// TIA Portal V21 export
TYPE "LAxisCtrl_typeGearOutCamOut"
TITLE = LAxisCtrl_typeGearOutCamOut
// Support: tech.team.motioncontrol@siemens.com
   STRUCT
      slavePosition : LReal := 0.0;   // Stop position of following axis
      syncProfileReference : DInt := 1;   // Type of desynchronization (0: Desynchronize using dynamic behavior; 1: Desynchronize using leading value distance; 5: Cancel only a pending gearing / camming)
      masterStopDistance : LReal := 0.0;   // Leading value distance when "SyncProfileReference" = 1
      deceleration : LReal := -1.0;   // Deceleration for desynchronization (Value > 0.0: The specified value is used; Value = 0.0: Not permitted; Value < 0.0: Use of the default value configured in the technology object) when "SyncProfileReference" = 0
      jerk : LReal := -1.0;   // Jerk for desynchronization (Value > 0.0: Smooth velocity profile, the specified value is used; Value = 0.0: Trapezoidal velocity profile; Value < 0.0: Use of the default value configured in the technology object) when "SyncProfileReference" = 0
      syncOutDirection : DInt := 3;   // Desynchronization direction (1: Positive direction; 2: Negative direction; 3: Current direction)
      gearOutCamOutMode : DInt := -1;   // -1: Automatic detection whether to use a MC_GearOut or MC_CamOut; 0: Use of MC_GearOut; 1: Use of MC_CamOut
   END_STRUCT;
END_TYPE
